// Mitsubishi GX Works2 project: FINAL 14.6   PLC: FX3G

// global labels: Global1
VAR_GLOBAL
  Start_Input AT X001 : BOOL;
  Analog_input1 AT D8280 : INT;
END_VAR
VAR_GLOBAL CONSTANT
  Div400 : REAL := 400;
  Const5 : REAL;
END_VAR
VAR_GLOBAL
  Regular_gummygum AT M1 : BOOL;
  Start_day AT X007 : BOOL;
  Check AT Y011 : BOOL;
END_VAR
VAR_GLOBAL CONSTANT
  Const_5 : REAL := 5.0;
  Const_10 : REAL := 10.0;
  Const_6 : REAL := 6.0;
END_VAR
VAR_GLOBAL
  Lemon_amount AT D1112 : REAL;
  Stabilizer_amount AT D1114 : REAL;
  GummyBears_amount AT D1116 : REAL;
  Lemon_input AT D1122 : REAL;
  Stabilizer_input AT D1124 : REAL;
  GummyBears_input AT D1126 : REAL;
END_VAR
VAR_GLOBAL CONSTANT
  Lemon_35 : REAL := 35.0;
  Stabilizer_35 : REAL := 35.0;
  Lemon_455 : REAL := 455.0;
  Stabilizer_105 : REAL := 105.0;
END_VAR
VAR_GLOBAL
  Icecream_in_Making AT Y000 : BOOL;
  TC_making_timer AT TC2 : BOOL;
END_VAR
VAR_GLOBAL CONSTANT
  Timer_5sec : INT := K50;
  Raspberry_quantity_280 : REAL := 280.0;
END_VAR
VAR_GLOBAL
  Raspberry_input AT D1108 : REAL;
END_VAR
VAR_GLOBAL CONSTANT
  test1 : REAL := 1000;
  test2 : REAL := 500;
  test13 : REAL := 1000;
END_VAR
VAR_GLOBAL
  TS_making_time AT TS2 : BOOL;
END_VAR
VAR_GLOBAL CONSTANT
  Raspberry_quantity_385 : REAL := 385;
  Lemon_665 : REAL := 665;
  Stabilizer_210 : REAL := 210.0;
END_VAR
VAR_GLOBAL
  Start_cooling AT X002 : BOOL;
  TC_cooling_timer AT TC3 : BOOL;
END_VAR
VAR_GLOBAL CONSTANT
  Timer_8sec : INT := K80;
END_VAR
VAR_GLOBAL
  TS_cooling_time AT TS3 : BOOL;
  Sensor_temp_in_cooling AT X003 : BOOL;
  TestLamp AT M99 : BOOL;
  Icecream_cooling AT Y002 : BOOL;
  Finished_Icecream_counter AT D7000 : REAL;
  Finished_inventory_regular AT M10 : BOOL;
  Finished_inventory_treat AT M11 : BOOL;
  Emeregency_case AT X005 : BOOL;
END_VAR
VAR_GLOBAL CONSTANT
  reset_0 : REAL;
END_VAR
VAR_GLOBAL
  Reset0 AT M81 : BOOL;
  Releasing_M1 AT M118 : BOOL;
  Holding_M2 AT M217 : BOOL;
  Releasing_M2 AT M218 : BOOL;
  Raspberry_icecream_container AT D1160 : REAL;
  Lemon_icecream_container AT D1162 : REAL;
END_VAR
VAR_GLOBAL CONSTANT
  Lemon_350 : REAL := 350;
  Raspberry_490 : REAL := 490;
  Raspberry_350 : REAL := 350;
  Lemon_490 : REAL := 490;
  Raspberry_560 : REAL := 560;
  Lemon_700 : REAL := 700;
END_VAR
VAR_GLOBAL
  Lemon_cooling_container AT D1166 : REAL;
  Raspberry_cooling_container AT D1164 : REAL;
  Raspberry_mixing_container AT D1170 : REAL;
  Lemon_mixing_container AT D1168 : REAL;
  Start_mixing_flag AT M9 : BOOL;
  Regular_flag AT M100 : BOOL;
  Treat_flag AT M200 : BOOL;
END_VAR
VAR_GLOBAL CONSTANT
  GummyBears_28 : REAL := 28;
  GummyBears_70 : REAL := 70;
END_VAR
VAR_GLOBAL
  Regular_Mixing_Time AT TC4 : BOOL;
END_VAR
VAR_GLOBAL CONSTANT
  Timer_3sec : INT := K30;
END_VAR
VAR_GLOBAL
  Treat_Mixing_Time AT TC5 : BOOL;
END_VAR
VAR_GLOBAL CONSTANT
  Timer_5_seconds : INT := K50;
END_VAR
VAR_GLOBAL
  TS_Regular_Mixing_Time AT TS4 : BOOL;
  TS_Treat_Mixing_Time AT TS5 : BOOL;
  Flashing_1 AT TC7 : BOOL;
END_VAR
VAR_GLOBAL CONSTANT
  Constant_Half_Second : INT := K5;
END_VAR
VAR_GLOBAL
  Icecream_in_mixing1 AT Y005 : BOOL;
  Icecream_in_mixing2 AT Y006 : BOOL;
  Holding_M100 AT M101 : BOOL;
  Releasing_M100 AT M102 : BOOL;
  Releasing_M200 AT M202 : BOOL;
  Holding_M200 AT M201 : BOOL;
  Raspberry_Amount_1 AT D1128 : REAL;
  Icecream_in_making_flag AT M5 : BOOL;
  Icecream_in_making_flag2 AT M6 : BOOL;
  TC_making_timer2 AT TC20 : BOOL;
  TS_making_time2 AT TS20 : BOOL;
  Start_regular_icecream_making AT M7 : BOOL;
  Start_treat_icecream_making AT M71 : BOOL;
  Finish_treat_phase1 AT M4 : BOOL;
  Finish_regular_phase1 AT M3 : BOOL;
  Finish_cooling_flag AT M13 : BOOL;
  Start_flashing AT M22 : BOOL;
END_VAR
VAR_GLOBAL CONSTANT
  Timer_half_sec : INT := 5;
END_VAR
VAR_GLOBAL
  Flashing_1_over AT TS7 : BOOL;
  Flashing2 AT TC8 : BOOL;
  Flashing2_over AT TS8 : BOOL;
  Mixing_in_progress_flag2 AT M21 : BOOL;
  Treat_gummygum AT M2 : BOOL;
  Mixed_container AT D1172 : REAL;
  Mixing_regular_timer AT TC9 : BOOL;
  Mixing_treat_timer AT TC10 : BOOL;
END_VAR
VAR_GLOBAL CONSTANT
  Timer_3_sec : DWORD := 30;
  Mixing_3sec : INT := K30;
  Mixing_5sec : INT := K50;
END_VAR
VAR_GLOBAL
  Finish_3_sec AT TS9 : BOOL;
  Finish_5_sec AT TS10 : BOOL;
  Start_packing AT X004 : BOOL;
  Start_packing_single AT X000 : BOOL;
  Icecream_in_packing AT Y004 : BOOL;
  Count_7packed AT CC1 : BOOL;
  Finish_7pack AT CS1 : BOOL;
END_VAR
VAR_GLOBAL CONSTANT
  Const_1 : REAL := 1;
  Restart : REAL;
  Const_455 : REAL := 455.0;
  Const_280 : REAL := 280;
  Const_105 : REAL := 105;
  Const_28 : REAL := 28;
END_VAR
VAR_GLOBAL
  Regular_raspberry_inventory AT M41 : BOOL;
  Regular_stabiliz_inventory AT M42 : BOOL;
  Regular_gummy_inventory AT M43 : BOOL;
END_VAR
VAR_GLOBAL CONSTANT
  Const_665 : REAL := 665;
END_VAR
VAR_GLOBAL
  Treat_lemon_inventory AT M44 : BOOL;
END_VAR
VAR_GLOBAL CONSTANT
  Const_385 : REAL := 385;
END_VAR
VAR_GLOBAL
  Treat_raspberry_inventory AT M45 : BOOL;
END_VAR
VAR_GLOBAL CONSTANT
  Const_210 : REAL := 210;
END_VAR
VAR_GLOBAL
  Treat_stabiliz_inventory AT M46 : BOOL;
END_VAR
VAR_GLOBAL CONSTANT
  Const_70 : REAL := 70;
END_VAR
VAR_GLOBAL
  Treat_gummy_inventory AT M47 : BOOL;
END_VAR
VAR_GLOBAL CONSTANT
  Const1 : REAL := 1.0;
END_VAR
VAR_GLOBAL
  Enough_regular_inventory AT M48 : BOOL;
  Finish_total_inventory AT M51 : BOOL;
  Day_hasnt_finished AT M52 : BOOL;
  ChecK_TEST_TEST AT M57 : BOOL;
  Start_working AT Y007 : BOOL;
END_VAR
VAR_GLOBAL CONSTANT
  Const_5ANDHALF : REAL := 5.0;
  Const_5_and_half : REAL := 5.0;
  Const_5_5 : REAL := 5.5;
  Const_6_5 : REAL := 6.5;
END_VAR
VAR_GLOBAL
  Enough_treat_inventory AT M58 : BOOL;
  Start_cooling_flagg AT M50 : BOOL;
  Finish_round_flag AT M72 : BOOL;
  Cooling_flag AT M73 : BOOL;
  Start_regular_making_flag AT M76 : BOOL;
  Start_treat_making_flag AT M78 : BOOL;
  Flag_finish_mixing_flag AT M79 : BOOL;
  seven_boom AT D1174 : INT;
END_VAR
VAR_GLOBAL CONSTANT
  Reset0_float : REAL;
  Const_4000 : REAL := 4000;
END_VAR
VAR_GLOBAL
  Finished_icecram_output AT D8282 : INT;
END_VAR
VAR_GLOBAL CONSTANT
  Const_40 : REAL := 40;
END_VAR

// task Task_01 (event TRUE, interval 0, priority 31): POU_01

PROGRAM POU_01
VAR CONSTANT
  Raspberry_280 : INT := K280;
END_VAR
VAR
  Temp_in_cooling_sensor : BOOL;
  Temp_in_cooling : BOOL;
  Raspberry_amount : BOOL;
END_VAR
VAR CONSTANT
  Counter_7 : INT := 7;
END_VAR
(* structured ladder/FBD written out as ST: instructions are called as NAME(EN, inputs, outputs); _pN, _eN, _tN stand for wires *)
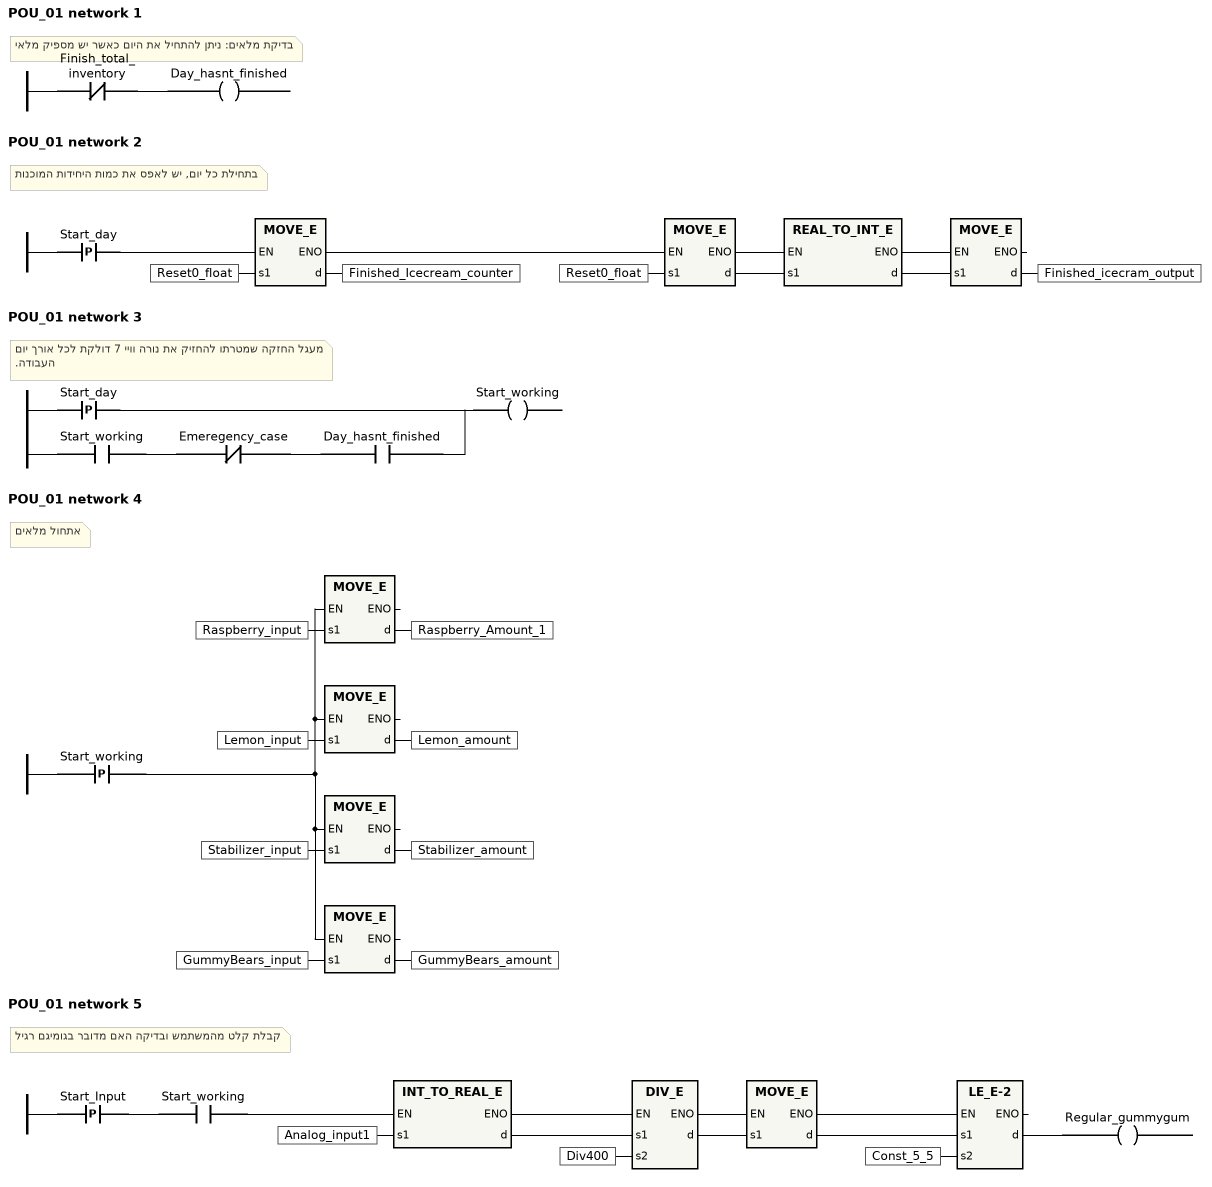
(* network 1 *)
(* בדיקת מלאים: ניתן להתחיל את היום כאשר יש מספיק מלאי *)
Day_hasnt_finished := NOT Finish_total_inventory;
(* network 2 *)
(* בתחילת כל יום, יש לאפס את כמות היחידות המוכנות *)
_e1 := MOVE_E(LDP(TRUE, Start_day), Reset0_float, Finished_Icecream_counter);
_e3 := MOVE_E(_e1, Reset0_float, _t2);
_e5 := REAL_TO_INT_E(_e3, _t2, _t4);
MOVE_E(_e5, _t4, Finished_icecram_output);
(* network 3 *)
(* מעגל החזקה שמטרתו להחזיק את נורה וויי 7 דולקת לכל אורך יום העבודה. *)
Start_working := LDP(TRUE, Start_day) OR (Start_working AND NOT Emeregency_case AND Day_hasnt_finished);
(* network 4 *)
(* אתחול מלאים *)
_p1 := LDP(TRUE, Start_working);
MOVE_E(_p1, Raspberry_input, Raspberry_Amount_1);
MOVE_E(_p1, Lemon_input, Lemon_amount);
MOVE_E(_p1, Stabilizer_input, Stabilizer_amount);
MOVE_E(_p1, GummyBears_input, GummyBears_amount);
(* network 5 *)
(* קבלת קלט מהמשתמש ובדיקה האם מדובר בגומיגם רגיל *)
_e2 := INT_TO_REAL_E(LDP(TRUE, Start_Input) AND Start_working, Analog_input1, _t1);
_e4 := DIV_E(_e2, _t1, Div400, _t3);
_e6 := MOVE_E(_e4, _t3, _t5);
LE_E(_e6, _t5, Const_5_5, _t7);
Regular_gummygum := _t7;
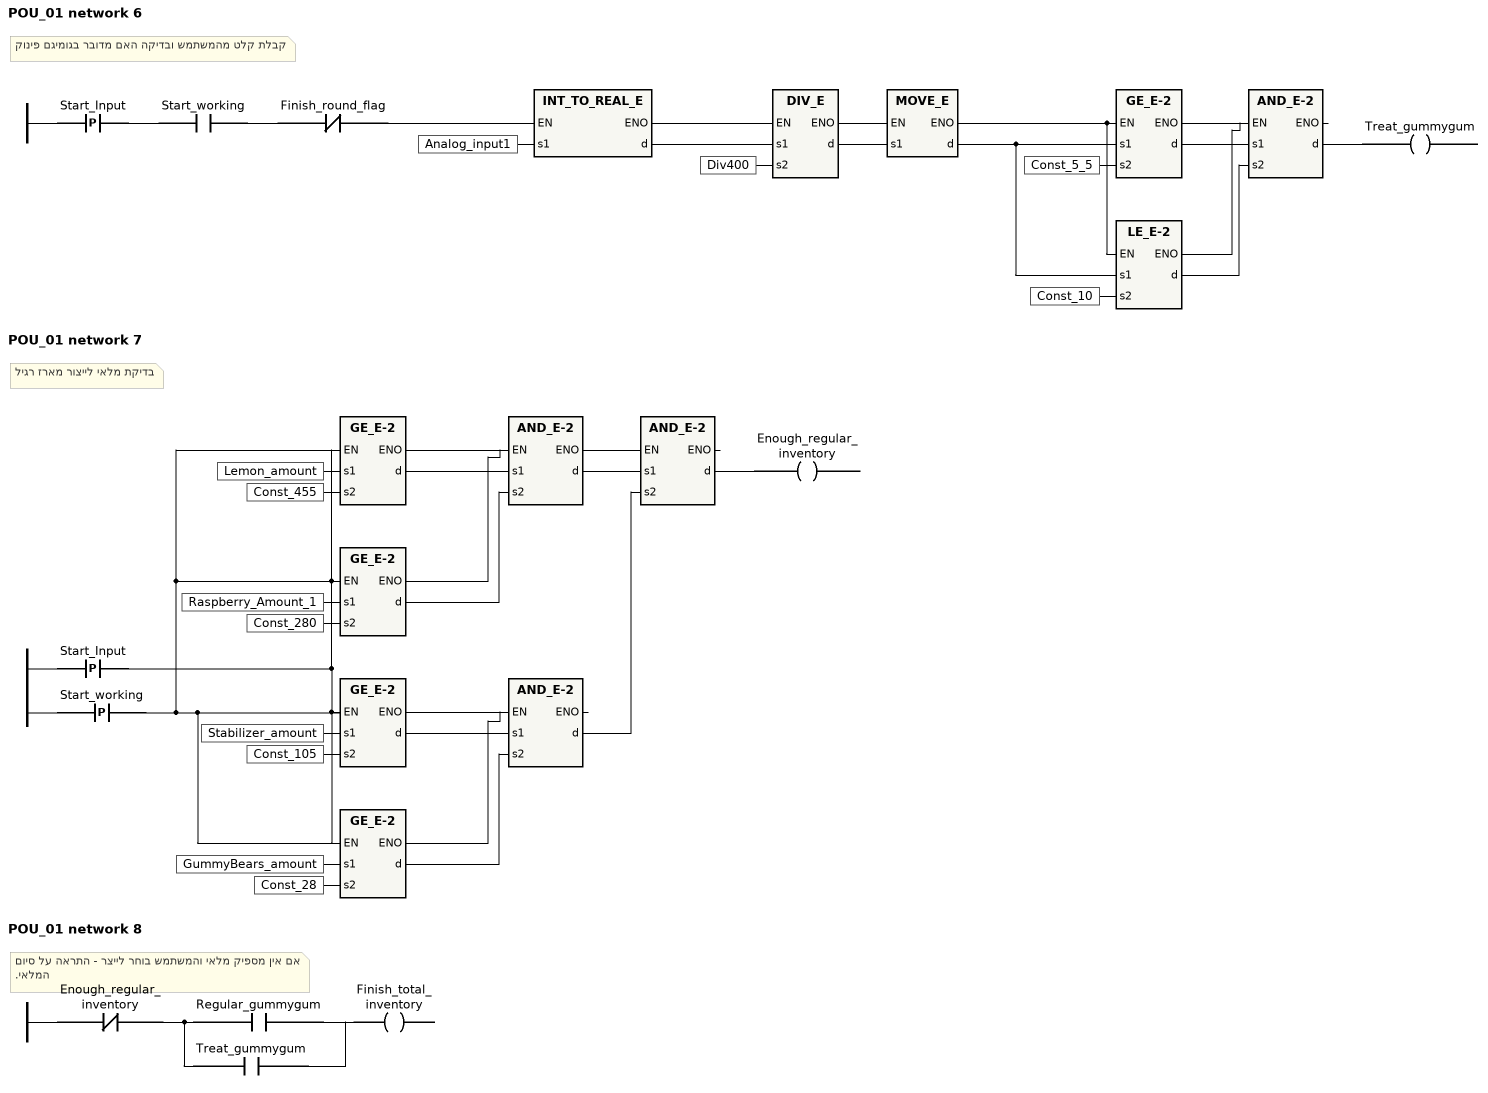
(* network 6 *)
(* קבלת קלט מהמשתמש ובדיקה האם מדובר בגומיגם פינוק *)
_e2 := INT_TO_REAL_E(LDP(TRUE, Start_Input) AND Start_working AND NOT Finish_round_flag, Analog_input1, _t1);
_e4 := DIV_E(_e2, _t1, Div400, _t3);
_e6 := MOVE_E(_e4, _t3, _t5);
_e8 := GE_E(_e6, _t5, Const_5_5, _t7);
_e10 := LE_E(_e6, _t5, Const_10, _t9);
AND_E(_e8 OR _e10, _t7, _t9, _t11);
Treat_gummygum := _t11;
(* network 7 *)
(* בדיקת מלאי לייצור מארז רגיל *)
_p1 := LDP(TRUE, Start_Input) OR LDP(TRUE, Start_working);
_e3 := GE_E(_p1, Lemon_amount, Const_455, _t2);
_e5 := GE_E(_p1, Raspberry_Amount_1, Const_280, _t4);
_e7 := AND_E(_e3 OR _e5, _t2, _t4, _t6);
_e9 := GE_E(_p1, Stabilizer_amount, Const_105, _t8);
_e11 := GE_E(_p1, GummyBears_amount, Const_28, _t10);
AND_E(_e9 OR _e11, _t8, _t10, _t12);
AND_E(_e7, _t6, _t12, _t13);
Enough_regular_inventory := _t13;
(* network 8 *)
(* אם אין מספיק מלאי והמשתמש בוחר לייצר - התראה על סיום המלאי. *)
_p1 := NOT Enough_regular_inventory;
Finish_total_inventory := (_p1 AND Regular_gummygum) OR (_p1 AND Treat_gummygum);
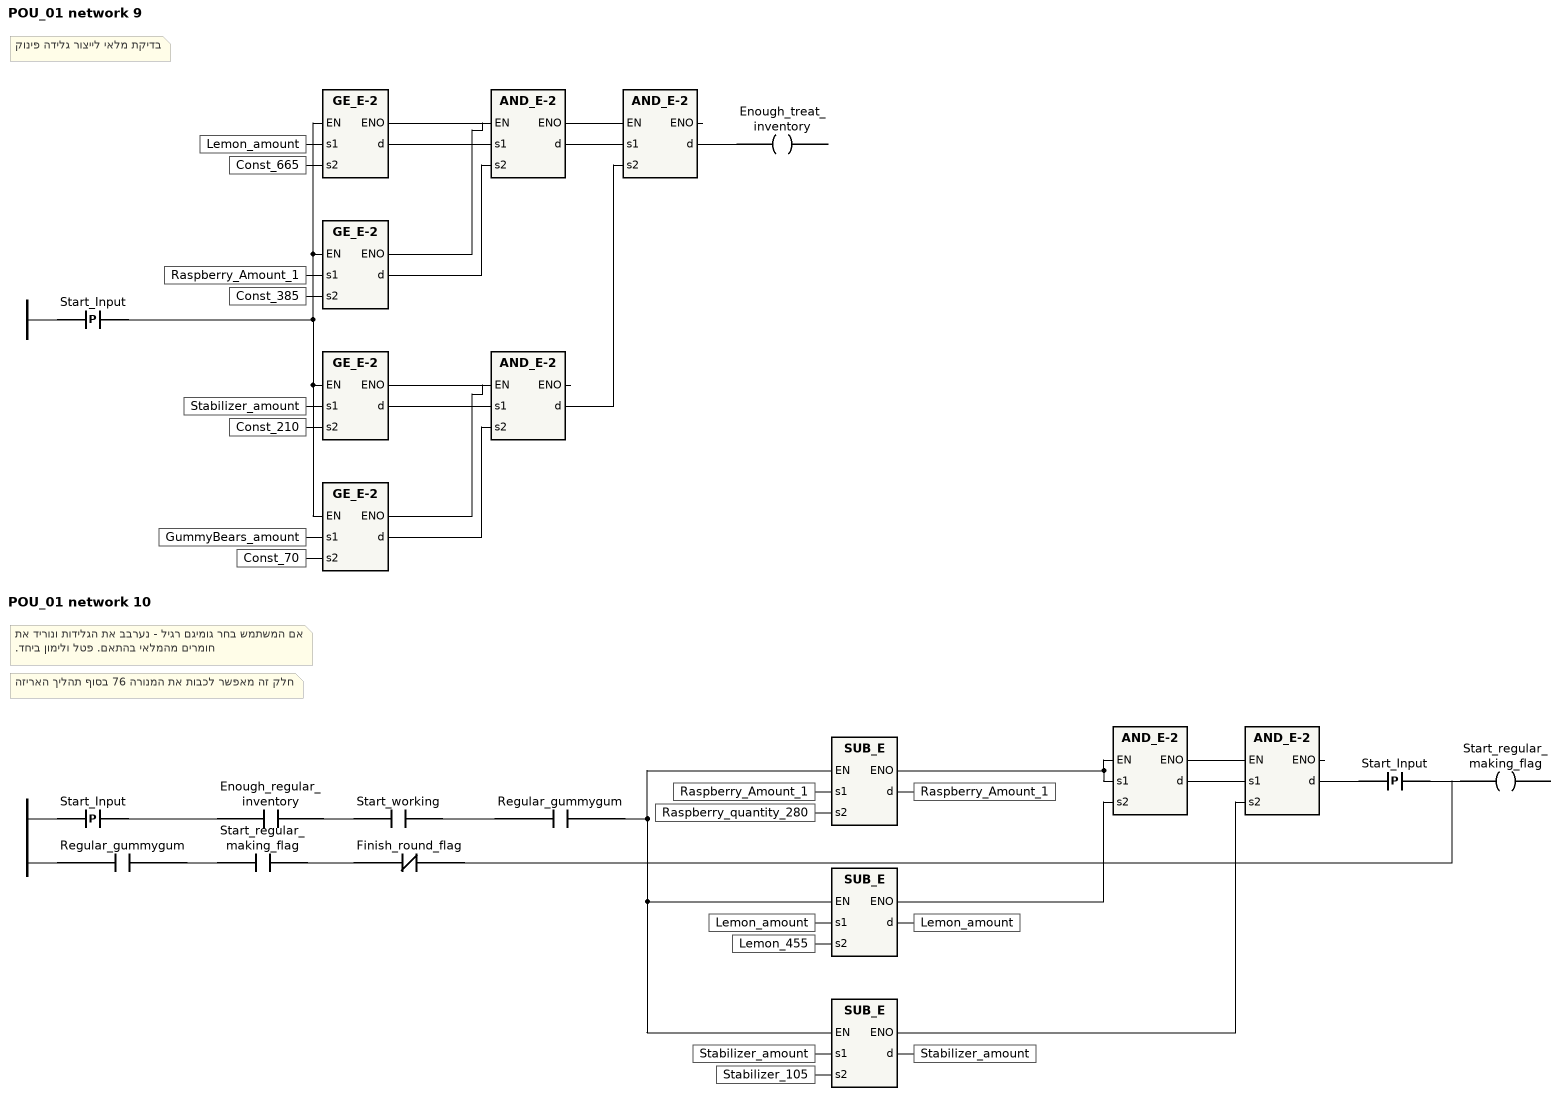
(* network 9 *)
(* בדיקת מלאי לייצור גלידה פינוק *)
_p1 := LDP(TRUE, Start_Input);
_e3 := GE_E(_p1, Lemon_amount, Const_665, _t2);
_e5 := GE_E(_p1, Raspberry_Amount_1, Const_385, _t4);
_e7 := AND_E(_e3 OR _e5, _t2, _t4, _t6);
_e9 := GE_E(_p1, Stabilizer_amount, Const_210, _t8);
_e11 := GE_E(_p1, GummyBears_amount, Const_70, _t10);
AND_E(_e9 OR _e11, _t8, _t10, _t12);
AND_E(_e7, _t6, _t12, _t13);
Enough_treat_inventory := _t13;
(* network 10 *)
(* אם המשתמש בחר גומיגם רגיל - נערבב את הגלידות ונוריד את חומרים מהמלאי בהתאם. פטל ולימון ביחד. *)
(* חלק זה מאפשר לכבות את המנורה 76 בסוף תהליך האריזה *)
_p1 := LDP(TRUE, Start_Input) AND Enough_regular_inventory AND Start_working AND Regular_gummygum;
_e2 := SUB_E(_p1, Raspberry_Amount_1, Raspberry_quantity_280, Raspberry_Amount_1);
_e3 := SUB_E(_p1, Lemon_amount, Lemon_455, Lemon_amount);
_e5 := AND_E(_e2, _e2, _e3, _t4);
_e6 := SUB_E(_p1, Stabilizer_amount, Stabilizer_105, Stabilizer_amount);
AND_E(_e5, _t4, _e6, _t7);
Start_regular_making_flag := (_t7 AND LDP(TRUE, Start_Input)) OR (Regular_gummygum AND Start_regular_making_flag AND NOT Finish_round_flag);
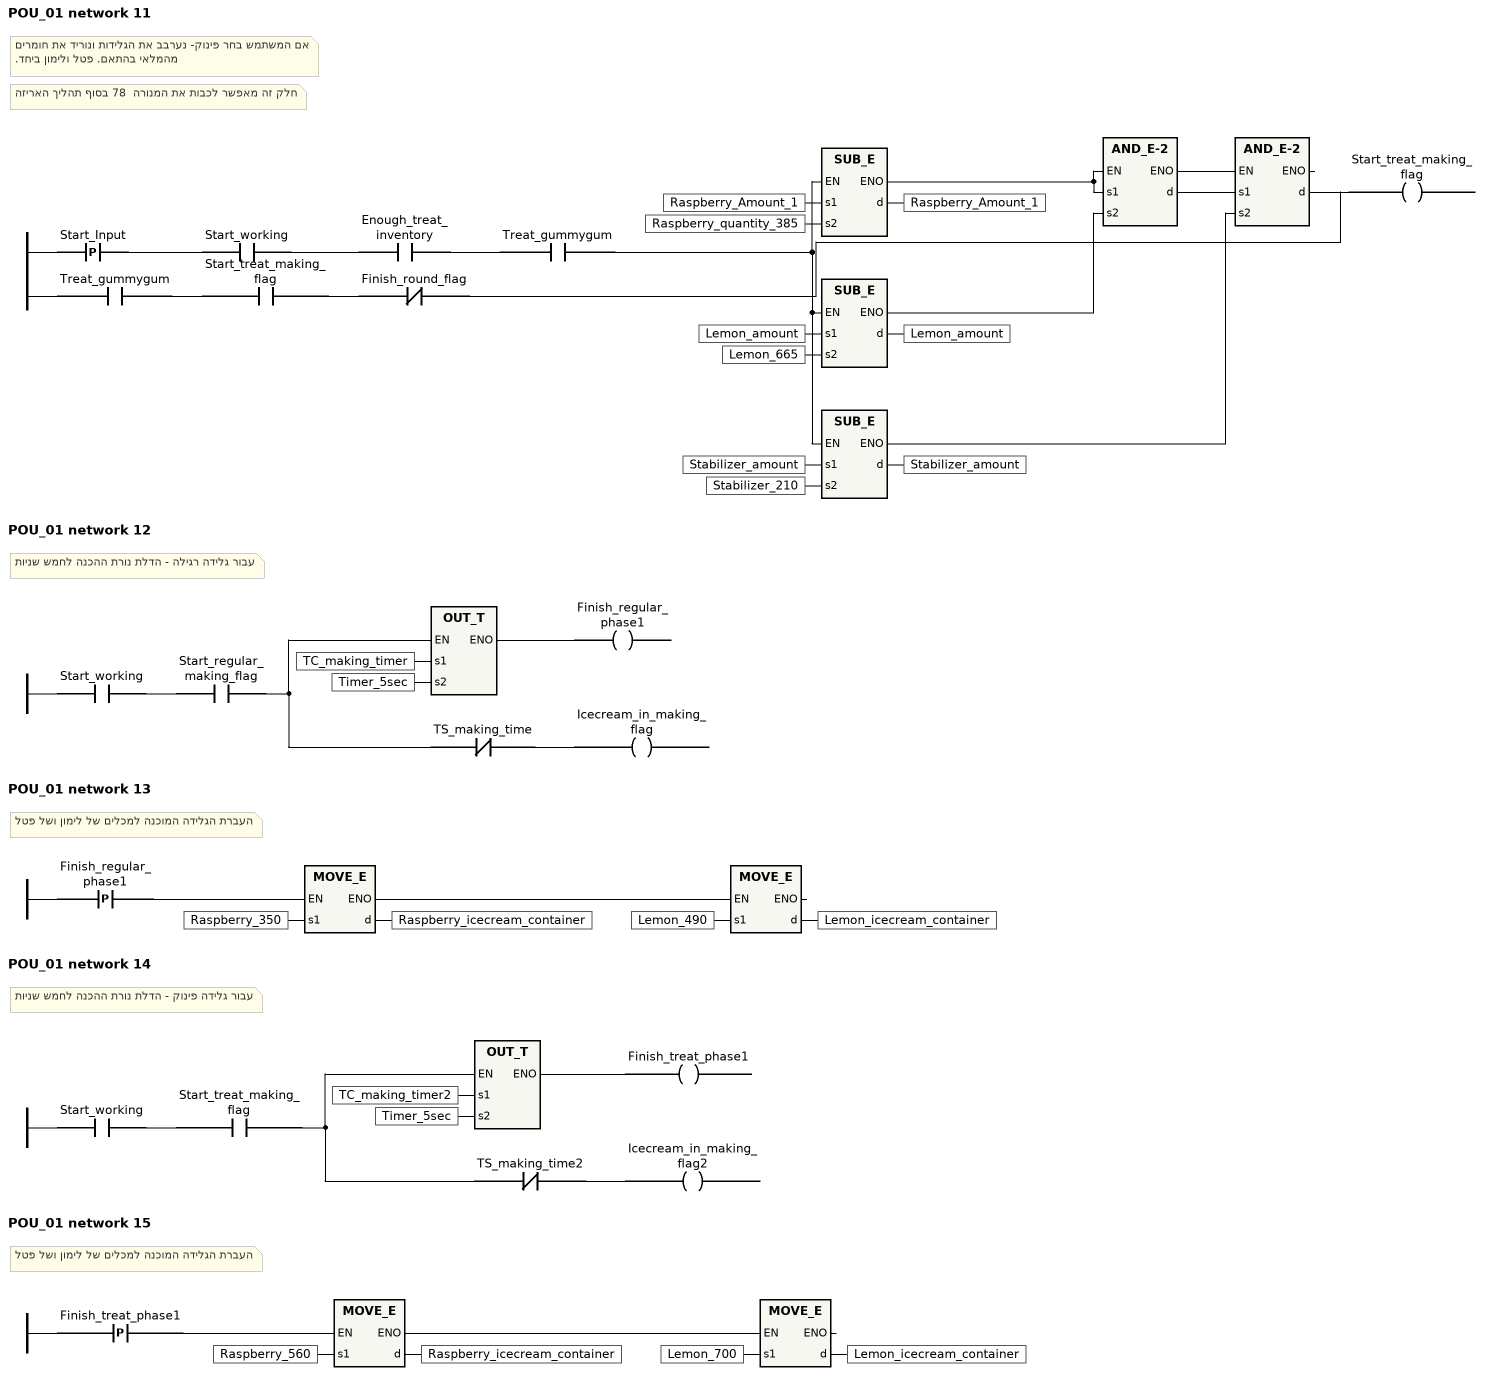
(* network 11 *)
(* אם המשתמש בחר פינוק- נערבב את הגלידות ונוריד את חומרים מהמלאי בהתאם. פטל ולימון ביחד. *)
(* חלק זה מאפשר לכבות את המנורה  78 בסוף תהליך האריזה *)
_p1 := LDP(TRUE, Start_Input) AND Start_working AND Enough_treat_inventory AND Treat_gummygum;
_e2 := SUB_E(_p1, Raspberry_Amount_1, Raspberry_quantity_385, Raspberry_Amount_1);
_e3 := SUB_E(_p1, Lemon_amount, Lemon_665, Lemon_amount);
_e5 := AND_E(_e2, _e2, _e3, _t4);
_e6 := SUB_E(_p1, Stabilizer_amount, Stabilizer_210, Stabilizer_amount);
AND_E(_e5, _t4, _e6, _t7);
Start_treat_making_flag := _t7 OR (Treat_gummygum AND Start_treat_making_flag AND NOT Finish_round_flag);
(* network 12 *)
(* עבור גלידה רגילה - הדלת נורת ההכנה לחמש שניות *)
_p1 := Start_working AND Start_regular_making_flag;
_e2 := OUT_T(_p1, TC_making_timer, Timer_5sec);
Finish_regular_phase1 := _e2;
Icecream_in_making_flag := _p1 AND NOT TS_making_time;
(* network 13 *)
(* העברת הגלידה המוכנה למכלים של לימון ושל פטל *)
_e1 := MOVE_E(LDP(TRUE, Finish_regular_phase1), Raspberry_350, Raspberry_icecream_container);
MOVE_E(_e1, Lemon_490, Lemon_icecream_container);
(* network 14 *)
(* עבור גלידה פינוק - הדלת נורת ההכנה לחמש שניות *)
_p1 := Start_working AND Start_treat_making_flag;
_e2 := OUT_T(_p1, TC_making_timer2, Timer_5sec);
Finish_treat_phase1 := _e2;
Icecream_in_making_flag2 := _p1 AND NOT TS_making_time2;
(* network 15 *)
(* העברת הגלידה המוכנה למכלים של לימון ושל פטל *)
_e1 := MOVE_E(LDP(TRUE, Finish_treat_phase1), Raspberry_560, Raspberry_icecream_container);
MOVE_E(_e1, Lemon_700, Lemon_icecream_container);
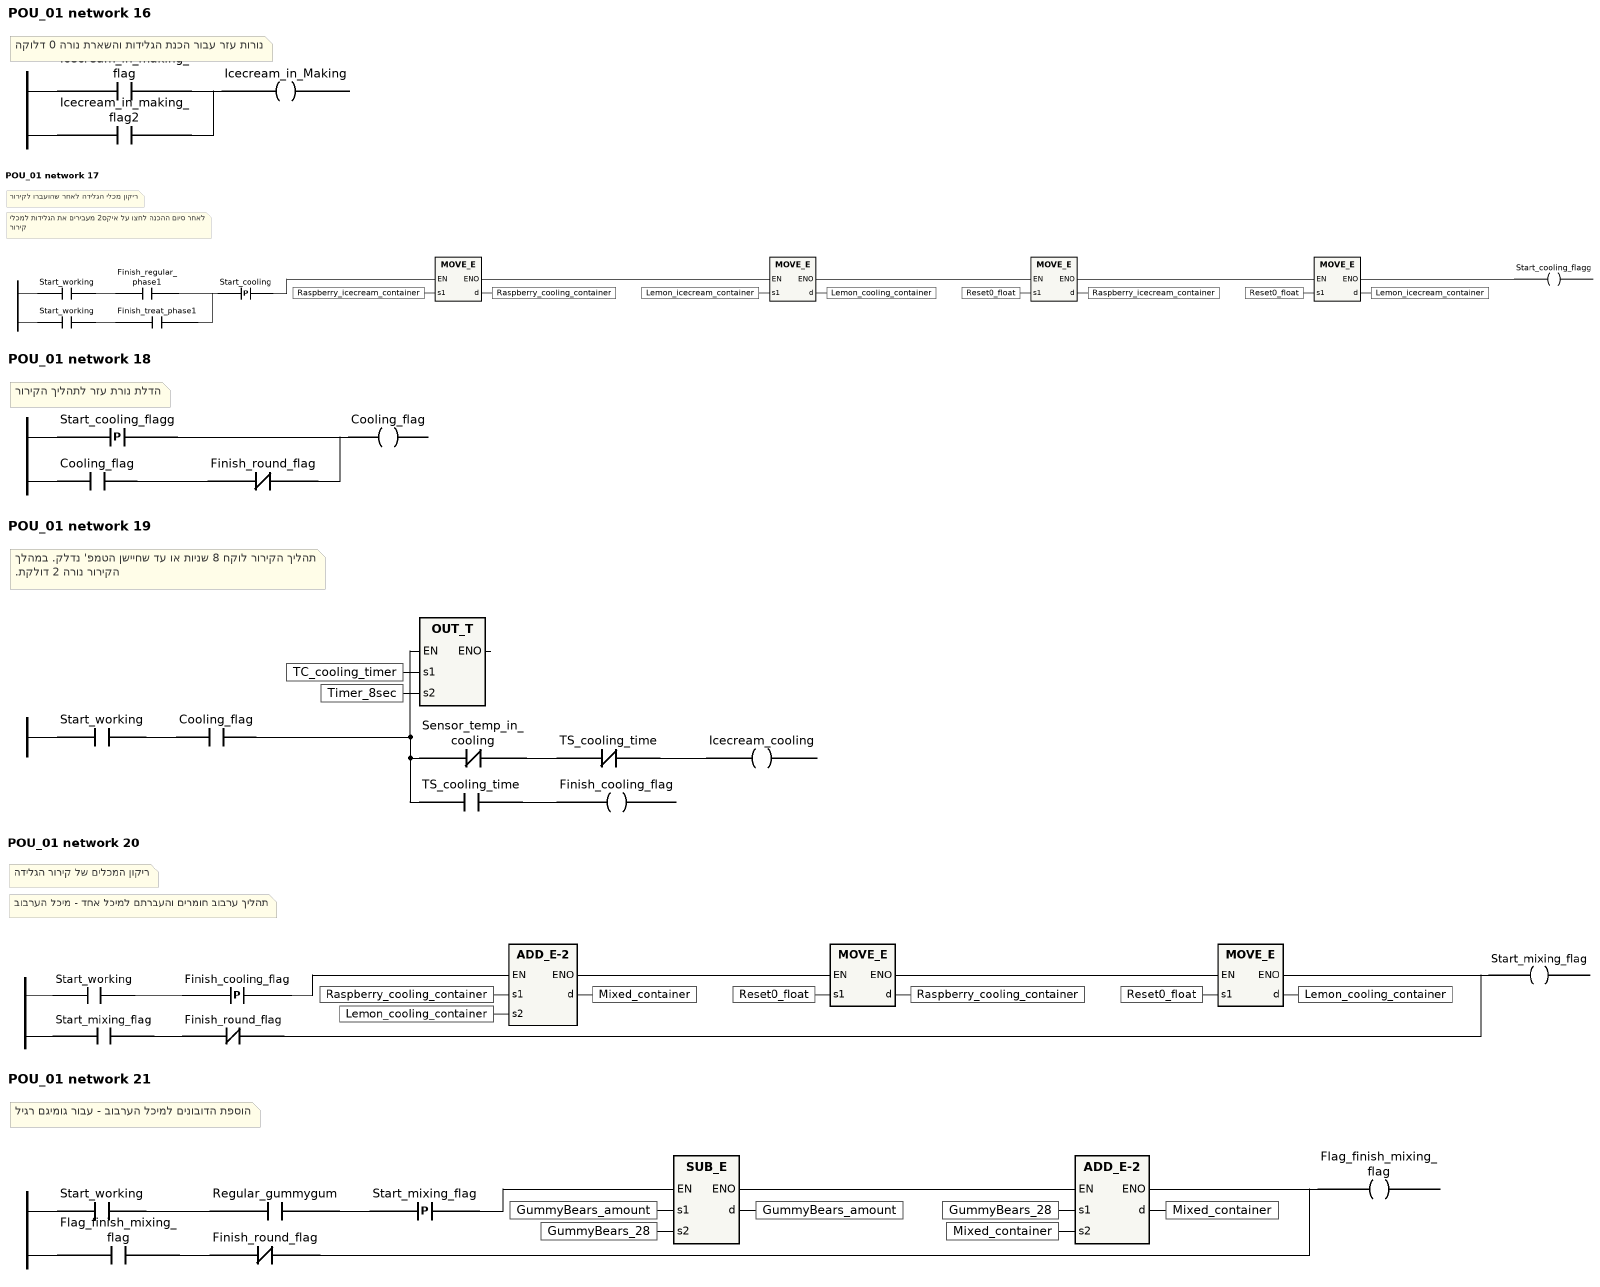
(* network 16 *)
(* נורות עזר עבור הכנת הגלידות והשארת נורה 0 דלוקה *)
Icecream_in_Making := Icecream_in_making_flag OR Icecream_in_making_flag2;
(* network 17 *)
(* ריקון מכלי הגלידה לאחר שהועברו לקירור *)
(* לאחר סיום ההכנה לחצו על איקס2 מעבירים את הגלידות למכלי קירור *)
_e1 := MOVE_E(((Start_working AND Finish_regular_phase1) OR (Start_working AND Finish_treat_phase1)) AND LDP(TRUE, Start_cooling), Raspberry_icecream_container, Raspberry_cooling_container);
_e2 := MOVE_E(_e1, Lemon_icecream_container, Lemon_cooling_container);
_e3 := MOVE_E(_e2, Reset0_float, Raspberry_icecream_container);
_e4 := MOVE_E(_e3, Reset0_float, Lemon_icecream_container);
Start_cooling_flagg := _e4;
(* network 18 *)
(* הדלת נורת עזר לתהליך הקירור *)
Cooling_flag := LDP(TRUE, Start_cooling_flagg) OR (Cooling_flag AND NOT Finish_round_flag);
(* network 19 *)
(* תהליך הקירור לוקח 8 שניות או עד שחיישן הטמפ' נדלק. במהלך הקירור נורה 2 דולקת. *)
_p1 := Start_working AND Cooling_flag;
OUT_T(_p1, TC_cooling_timer, Timer_8sec);
Icecream_cooling := _p1 AND NOT Sensor_temp_in_cooling AND NOT TS_cooling_time;
Finish_cooling_flag := _p1 AND TS_cooling_time;
(* network 20 *)
(* ריקון המכלים של קירור הגלידה *)
(* תהליך ערבוב חומרים והעברתם למיכל אחד - מיכל הערבוב *)
_e1 := ADD_E(Start_working AND LDP(TRUE, Finish_cooling_flag), Raspberry_cooling_container, Lemon_cooling_container, Mixed_container);
_e2 := MOVE_E(_e1, Reset0_float, Raspberry_cooling_container);
_e3 := MOVE_E(_e2, Reset0_float, Lemon_cooling_container);
Start_mixing_flag := _e3 OR (Start_mixing_flag AND NOT Finish_round_flag);
(* network 21 *)
(* הוספת הדובונים למיכל הערבוב - עבור גומיגם רגיל *)
_e1 := SUB_E(Start_working AND Regular_gummygum AND LDP(TRUE, Start_mixing_flag), GummyBears_amount, GummyBears_28, GummyBears_amount);
_e2 := ADD_E(_e1, GummyBears_28, Mixed_container, Mixed_container);
Flag_finish_mixing_flag := _e2 OR (Flag_finish_mixing_flag AND NOT Finish_round_flag);
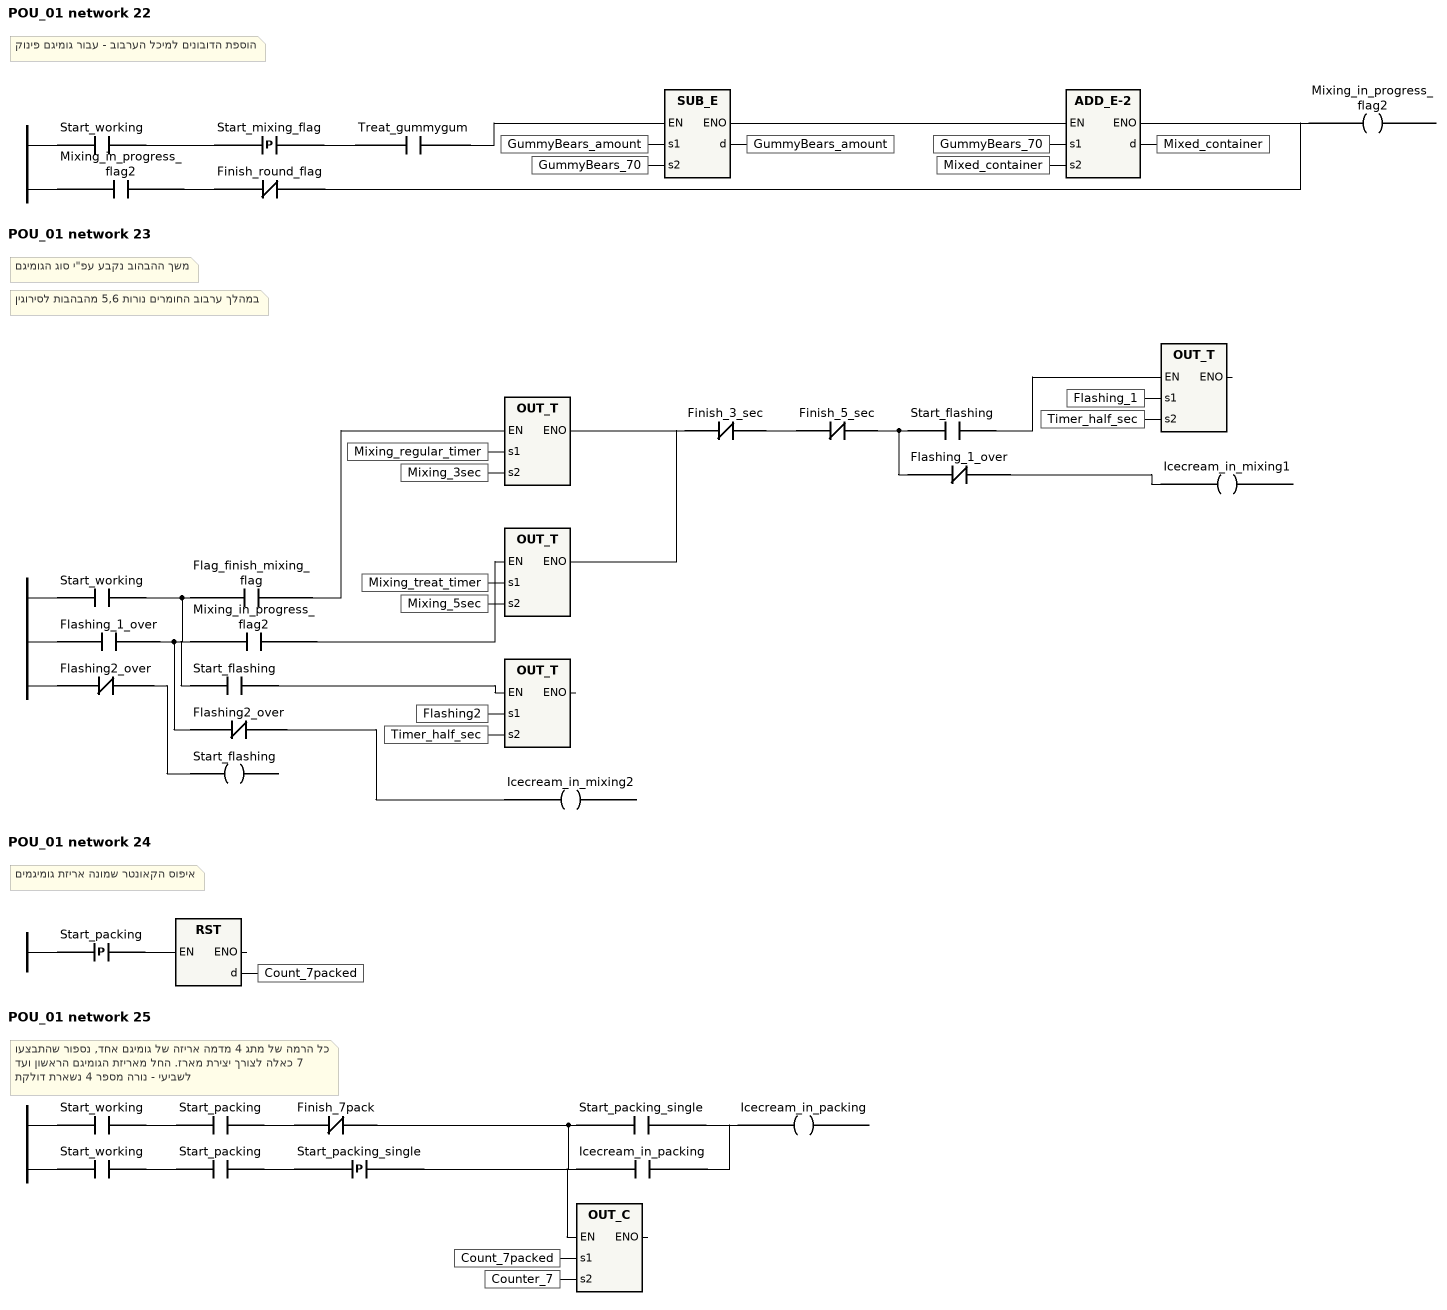
(* network 22 *)
(* הוספת הדובונים למיכל הערבוב - עבור גומיגם פינוק *)
_e1 := SUB_E(Start_working AND LDP(TRUE, Start_mixing_flag) AND Treat_gummygum, GummyBears_amount, GummyBears_70, GummyBears_amount);
_e2 := ADD_E(_e1, GummyBears_70, Mixed_container, Mixed_container);
Mixing_in_progress_flag2 := _e2 OR (Mixing_in_progress_flag2 AND NOT Finish_round_flag);
(* network 23 *)
(* משך ההבהוב נקבע עפ"י סוג הגומיגם *)
(* במהלך ערבוב החומרים נורות 5,6 מהבהבות לסירוגין *)
_e1 := OUT_T(Start_working AND Flag_finish_mixing_flag, Mixing_regular_timer, Mixing_3sec);
_e2 := OUT_T(Start_working AND Mixing_in_progress_flag2, Mixing_treat_timer, Mixing_5sec);
_p3 := ((_e1 OR _e2) AND NOT Finish_3_sec) AND NOT Finish_5_sec;
OUT_T(_p3 AND Start_flashing, Flashing_1, Timer_half_sec);
Icecream_in_mixing1 := _p3 AND NOT Flashing_1_over;
OUT_T(Flashing_1_over AND Start_flashing, Flashing2, Timer_half_sec);
Icecream_in_mixing2 := Flashing_1_over AND NOT Flashing2_over;
Start_flashing := NOT Flashing2_over;
(* network 24 *)
(* איפוס הקאונטר שמונה אריזת גומיגמים *)
RST(LDP(TRUE, Start_packing), Count_7packed);
(* network 25 *)
(* כל הרמה של מתג 4 מדמה אריזה של גומיגם אחד, נספור שהתבצעו 7 כאלה לצורך יצירת מארז. החל מאריזת הגומיגם הראשון ועד לשביעי - נורה מספר 4 נשארת דולקת *)
_p1 := Start_working AND Start_packing AND NOT Finish_7pack;
Icecream_in_packing := (_p1 AND Start_packing_single) OR (_p1 AND Icecream_in_packing);
OUT_C(Start_working AND Start_packing AND LDP(TRUE, Start_packing_single), Count_7packed, Counter_7);
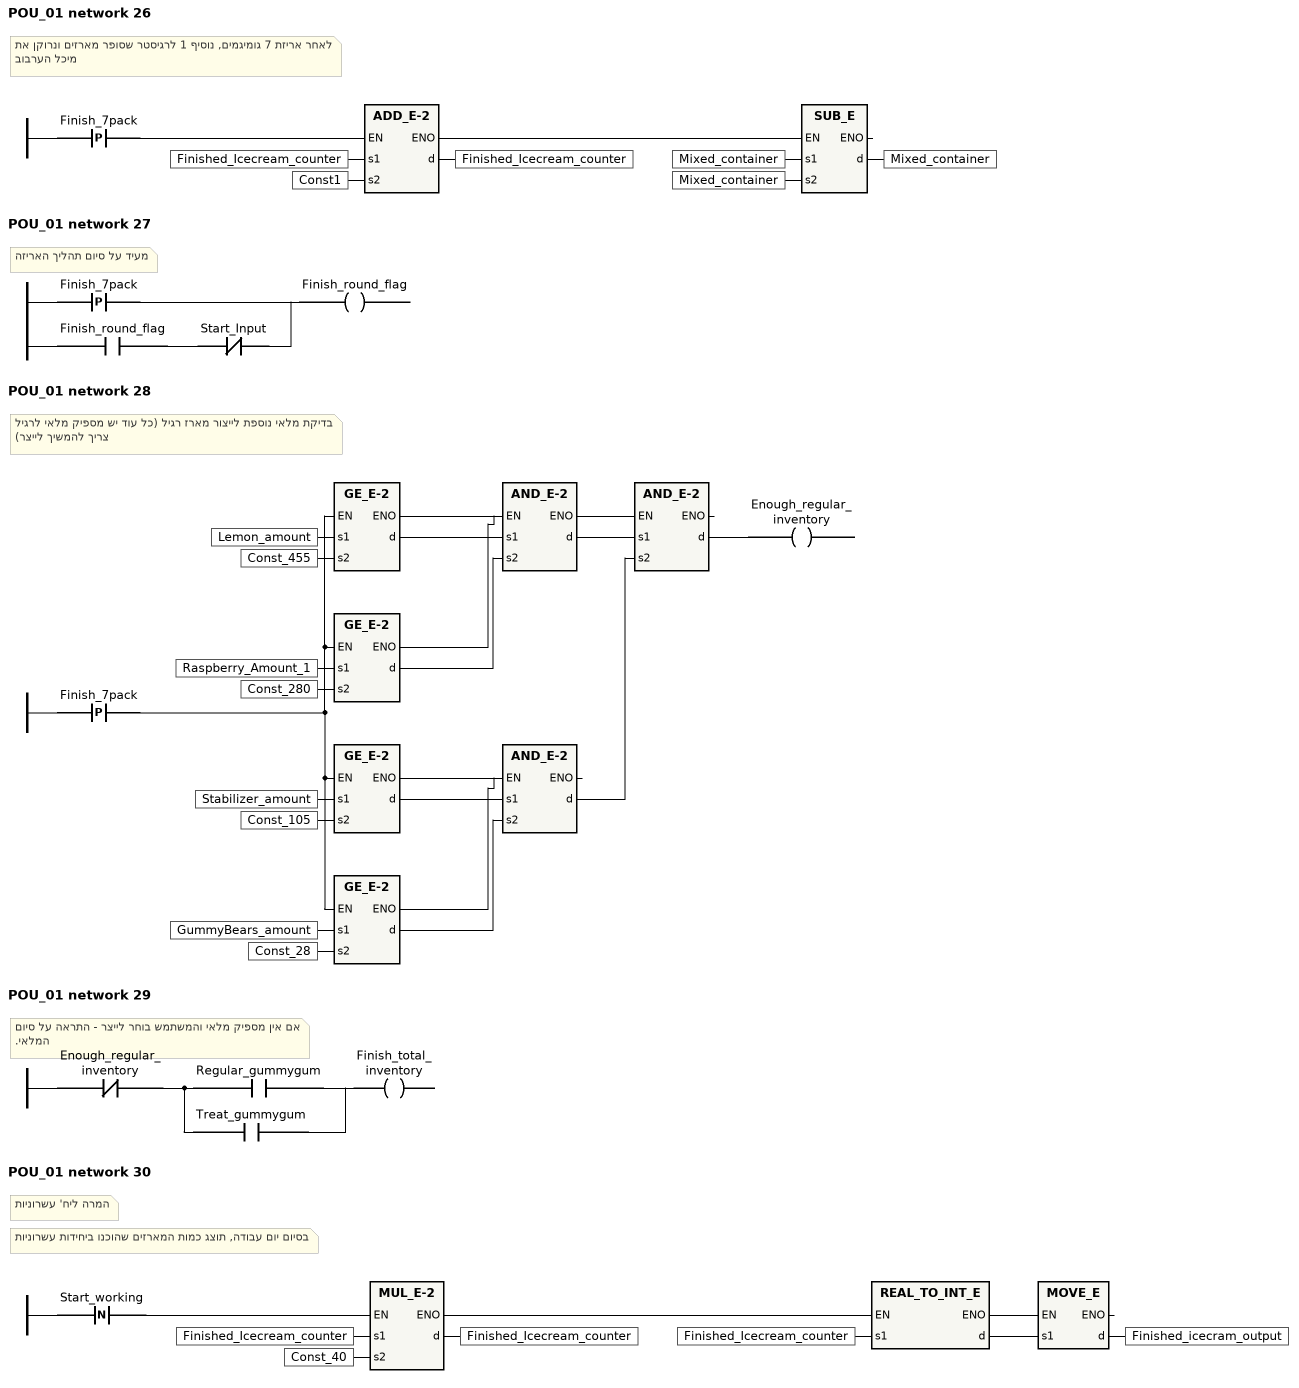
(* network 26 *)
(* לאחר אריזת 7 גומיגמים, נוסיף 1 לרגיסטר שסופר מארזים ונרוקן את מיכל הערבוב *)
_e1 := ADD_E(LDP(TRUE, Finish_7pack), Finished_Icecream_counter, Const1, Finished_Icecream_counter);
SUB_E(_e1, Mixed_container, Mixed_container, Mixed_container);
(* network 27 *)
(* מעיד על סיום תהליך האריזה *)
Finish_round_flag := LDP(TRUE, Finish_7pack) OR (Finish_round_flag AND NOT Start_Input);
(* network 28 *)
(* בדיקת מלאי נוספת לייצור מארז רגיל (כל עוד יש מספיק מלאי לרגיל צריך להמשיך לייצר) *)
_p1 := LDP(TRUE, Finish_7pack);
_e3 := GE_E(_p1, Lemon_amount, Const_455, _t2);
_e5 := GE_E(_p1, Raspberry_Amount_1, Const_280, _t4);
_e7 := AND_E(_e3 OR _e5, _t2, _t4, _t6);
_e9 := GE_E(_p1, Stabilizer_amount, Const_105, _t8);
_e11 := GE_E(_p1, GummyBears_amount, Const_28, _t10);
AND_E(_e9 OR _e11, _t8, _t10, _t12);
AND_E(_e7, _t6, _t12, _t13);
Enough_regular_inventory := _t13;
(* network 29 *)
(* אם אין מספיק מלאי והמשתמש בוחר לייצר - התראה על סיום המלאי. *)
_p1 := NOT Enough_regular_inventory;
Finish_total_inventory := (_p1 AND Regular_gummygum) OR (_p1 AND Treat_gummygum);
(* network 30 *)
(* המרה ליח' עשרוניות *)
(* בסיום יום עבודה, תוצג כמות המארזים שהוכנו ביחידות עשרוניות *)
_e1 := MUL_E(LDF(TRUE, Start_working), Finished_Icecream_counter, Const_40, Finished_Icecream_counter);
_e3 := REAL_TO_INT_E(_e1, Finished_Icecream_counter, _t2);
MOVE_E(_e3, _t2, Finished_icecram_output);
END_PROGRAM
